// TIA Portal V17 export
// export: Created 2021-12-03T08:12:58.5326538Z, ExportSetting WithDefaults, DisplayName Totally Integrated Automation Portal, DisplayVersion V17, DisplayName TIA Portal Openness, DisplayVersion V17, DisplayName TIA Portal Version Control Interface, DisplayVersion V17, DisplayName STEP 7 Professional, DisplayVersion V17, DisplayName STEP 7 Safety, DisplayVersion V17, DisplayName WinCC Advanced, DisplayVersion V17
ORGANIZATION_BLOCK "MOD_ERR"   // OB122, FBD, IOAccessError
TITLE = "Module Access Error"
VERSION : 0.1
// stored: IsIECCheckEnabled false
   VAR_TEMP
      OB122_EV_CLASS : Byte;   // 16#29, Event class 2, Entering event state, Internal fault event
      OB122_SW_FLT : Byte;   // 16#XX Software error code
      OB122_PRIORITY : Byte;   // Priority of OB Execution
      OB122_OB_NUMBR : Byte;   // 122 (Organization block 122, OB122)
      OB122_BLK_TYPE : Byte;   // 16#88/8C/8E Type of block fault occured in
      OB122_MEM_AREA : Byte;   // Memory area where access error occured
      OB122_MEM_ADDR : Word;   // Memory address where access error occured
      OB122_BLK_NUM : Word;   // Block number in which error occured
      OB122_PRG_ADDR : Word;   // Program address where error occured
      OB122_DATE_TIME : Date_And_Time;   // Date and time OB1 started
   END_VAR
BEGIN
END_ORGANIZATION_BLOCK
